// TwinCAT 3 PLC project SPS_Blinker
// ProgramVersion: 3.1.4026.19
// libraries:
//   Tc2_Standard, * (Beckhoff Automation GmbH)
//   Tc2_System, * (Beckhoff Automation GmbH)
//   Tc2_Utilities, * (Beckhoff Automation GmbH)
// project tree:
//   DUTs/ st_Data.TcDUT, ST_MyData.TcDUT, U_Convert.TcDUT, U_Convert_REAL.TcDUT
//   GVLs/ GVL.TcGVL, GVL_Blinker.TcGVL
//   GVLs/Temperaturfuehler/ GVL_Temperatur.TcGVL
//   / PlcTask.TcTTO
//   POUs/ alle_5sekunden.TcPOU, Blinker.TcPOU, LineChart.TcPOU, Line_Chart_array.TcPOU, MAIN.TcPOU, Modbus_Register_lesen.TcPOU, Modbus_Register_schreiben.TcPOU, Systemzeit.TcPOU, TOF_Beispiel.TcPOU
//   POUs/Funktionen_u_Bausteine/ FB_Blinker.TcPOU, FB_RWA_Trend_array.TcPOU
// real-time tasks:
//   TASK PlcTask: cycle T#10ms, priority 20, ADS port 350

CONFIGURATION SPS_Blinker
    RESOURCE PLC ON TwinCAT3
        TASK PlcTask(INTERVAL := T#10ms, PRIORITY := 20);
        PROGRAM MAIN WITH PlcTask : MAIN;
    END_RESOURCE
END_CONFIGURATION

// ---- DUTs/st_Data.TcDUT
TYPE st_Data :
STRUCT
	x	: INT;
	y	: INT;
END_STRUCT
END_TYPE

// ---- DUTs/ST_MyData.TcDUT
TYPE ST_MyData :
STRUCT
	Nr		: DINT;
	Zeit 	: DT;
	Wert 	: INT;
END_STRUCT
END_TYPE

// ---- DUTs/U_Convert.TcDUT
TYPE U_Convert :
UNION
	AsWord: ARRAY[0..1] OF WORD;
	AsReal: REAL;
END_UNION
END_TYPE

// ---- DUTs/U_Convert_REAL.TcDUT
TYPE U_Convert_REAL :
UNION
	AsReal: ARRAY[0..1] OF REAL;
	AsWord: WORD;
END_UNION
END_TYPE

// ---- GVLs/GVL.TcGVL
VAR_GLOBAL
	//Systemzeit
	bValid     			: BOOL := FALSE;
	
	dtsystemTime		: DATE_AND_TIME;
	
	todsystemTime		: TIME_OF_DAY;
	
	sAktuelle_Stunde	: STRING(255);	//Aktuelle Stunde als String
	
	iAktuelle_Stunde	: INT;			//Aktuelle Stunde als INT
	
	sAktuelle_Minute	: STRING(255);	//Aktuelle Minute als String
	
	iAktuelle_Minute	: INT;			//Aktuelle Minute als INT
	
	sAktuelle_Sekunde	: STRING(255);	//Aktuelle Sekunde als String
	
	iAktuelle_Sekunde	: INT;			//Aktuelle Sekunde als INT
	
	//Main
	bStartUpFinish		: BOOL;
END_VAR

// ---- GVLs/GVL_Blinker.TcGVL
VAR_GLOBAL
	rStatus		: REAL;
	bBlink		: BOOL;
END_VAR

// ---- GVLs/Temperaturfuehler/GVL_Temperatur.TcGVL
VAR_GLOBAL
//	rH0_Aussentemp_old	: REAL;	//Aussenfühler H0 Überdachung
	rH0_Aussentemp		: REAL;	//Aussenfühler H0 Überdachung
END_VAR

// ---- POUs/MAIN.TcPOU
PROGRAM MAIN
VAR

END_VAR

Systemzeit();
Blinker();
//Line_Chart_array();

//LineChart();
//TOF_Beispiel();

alle_5sekunden();

END_PROGRAM

// ---- POUs/Systemzeit.TcPOU
PROGRAM Systemzeit
VAR
	fbFB_LocalSystemTime: FB_LocalSystemTime;
	fbGETSYSTEMTIME		: GETSYSTEMTIME;
    sNetID     			: T_AmsNetID := '';
    bEnable    			: BOOL := 1;
    dwCycle    			: DWORD(1..86400) := 5;
    dwOpt      			: DWORD := 1;
    tTimeout   			: TIME := DEFAULT_ADS_TIMEOUT;
	//bValid     		: BOOL := FALSE; GVL
	//dtsystemTime		: DATE_AND_TIME; GVL
	tzID       			: E_TimeZoneID := eTimeZoneID_Invalid;
END_VAR
VAR_INPUT
    systemTime 			: TIMESTRUCT;
END_VAR
VAR_OUTPUT
	
END_VAR

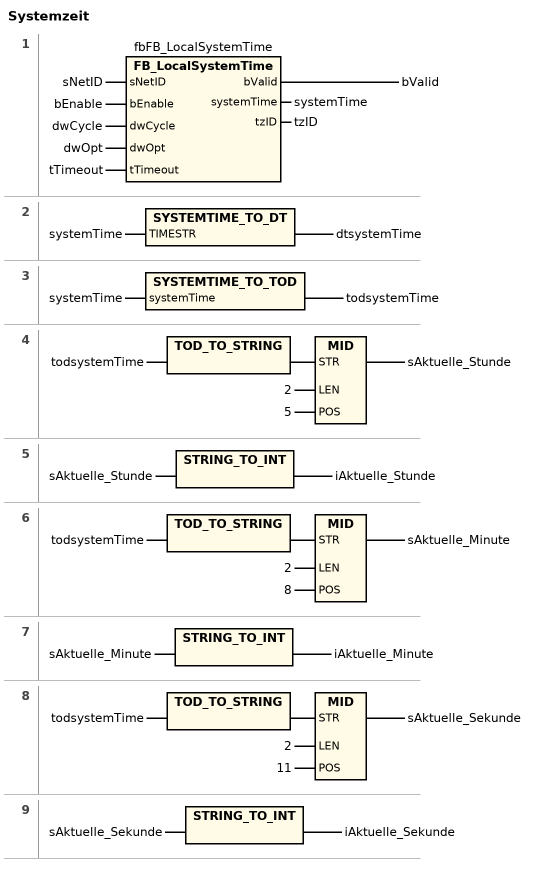
// NETWORK 1
fbFB_LocalSystemTime(
    sNetID := sNetID,
    bEnable := bEnable,
    dwCycle := dwCycle,
    dwOpt := dwOpt,
    tTimeout := tTimeout,
    systemTime => systemTime,
    tzID => tzID); // FB_LocalSystemTime
bValid := fbFB_LocalSystemTime.bValid;

// NETWORK 2
dtsystemTime := SYSTEMTIME_TO_DT(TIMESTR := systemTime);

// NETWORK 3
todsystemTime := SYSTEMTIME_TO_TOD(systemTime := systemTime);

// NETWORK 4
sAktuelle_Stunde := MID(STR := TOD_TO_STRING(todsystemTime), LEN := 2, POS := 5);

// NETWORK 5
iAktuelle_Stunde := STRING_TO_INT(sAktuelle_Stunde);

// NETWORK 6
sAktuelle_Minute := MID(STR := TOD_TO_STRING(todsystemTime), LEN := 2, POS := 8);

// NETWORK 7
iAktuelle_Minute := STRING_TO_INT(sAktuelle_Minute);

// NETWORK 8
sAktuelle_Sekunde := MID(STR := TOD_TO_STRING(todsystemTime), LEN := 2, POS := 11);

// NETWORK 9
iAktuelle_Sekunde := STRING_TO_INT(sAktuelle_Sekunde);

END_PROGRAM

// ---- POUs/Blinker.TcPOU
PROGRAM Blinker
VAR
	fbMyBlinker	: FB_Blinker;
//	bBlink		: BOOL;
END_VAR


fbMyBlinker(tBlinkOn:= T#500MS, tBlinkOff:=T#3S);
bBlink	:= fbMyBlinker.Q;

IF bBlink = TRUE THEN
	rStatus	:= 1;
ELSE	
	rStatus	:= 0;
END_IF

END_PROGRAM

// ---- POUs/Funktionen_u_Bausteine/FB_Blinker.TcPOU
FUNCTION_BLOCK FB_Blinker
VAR_INPUT
	tBlinkOn, tBlinkOff	: TIME;
END_VAR
VAR_OUTPUT
	Q	: BOOL;
END_VAR
VAR
	timerOn, timerOff	: TON;
	nState	: INT;
END_VAR

CASE nState OF
	0:		//Blinker on
		timerOn(IN:= TRUE,	PT:=tBlinkOn);
		Q	:= TRUE;
		IF timerOn.Q THEN
			timerOn(IN:=FALSE);
			nState := 1;
		END_IF
	1:		//Blinker off
		timerOff(IN:=TRUE, PT:=tBlinkOff);
		Q	:= FALSE;
		IF timerOff.Q THEN
			timerOff(IN:=FALSE);
			nState := 0;
		END_IF
END_CASE

END_FUNCTION_BLOCK

// ---- POUs/alle_5sekunden.TcPOU
PROGRAM alle_5sekunden
VAR
    arrData : ARRAY[1..10] OF REAL; // Beispiel-Array
    iSum : REAL;
    iAverage : REAL;
    i : INT;
	
END_VAR

// Summe der Elemente berechnen
iSum := 0;
FOR i := 1 TO 10 DO
    iSum := iSum + arrData[i];
END_FOR

// Durchschnitt berechnen (Division durch die Anzahl der Elemente)
//IF 10 > 0 THEN // Prüfen, ob die Anzahl der Elemente größer als 0 ist
    iAverage := iSum / 10; 
//END_IF

END_PROGRAM

// ---- POUs/Funktionen_u_Bausteine/FB_RWA_Trend_array.TcPOU
FUNCTION_BLOCK FB_RWA_Trend_array
VAR_IN_OUT
	aArray	: ARRAY[0..2,1..1000] OF ST_H2_4_trend_array;	
END_VAR
VAR_INPUT
	bFreigabe			: BOOL;
	rTrueWert			: REAL;
	rFalseWert			: REAL;	
	iArray_i			: DINT := 1;
	bFreigabe_save		: BOOL;	
END_VAR
VAR_OUTPUT
	iArray_i_out		: DINT;
	bFreigabe_save_out	: BOOL;	
END_VAR
VAR
	bEinmallauf			: BOOL;
END_VAR

IF bEinmallauf = FALSE THEN
		IF bFreigabe = TRUE THEN
				aArray[0,iArray_i].Nr	:= iArray_i;	//Laufende Nr
				aArray[0,iArray_i].Zeit	:= dtsystemTime;//Zeit
				aArray[0,iArray_i].Wert	:= rTrueWert;	//Wert Chart
			ELSE
				aArray[0,iArray_i].Nr	:= iArray_i;	//Laufende Nr
				aArray[0,iArray_i].Zeit	:= dtsystemTime;//Zeit
				aArray[0,iArray_i].Wert	:= rFalseWert;	//Wert Chart
		END_IF	
	iArray_i := (iArray_i+1);
	bEinmallauf := TRUE;
END_IF

IF (bFreigabe <> bFreigabe_save) THEN 
		IF bFreigabe = TRUE THEN
				//Zuerst den alten Wert schreiben damit der Chart waagrecht bleibt
				aArray[0,iArray_i].Nr	:= iArray_i;
				aArray[0,iArray_i].Zeit	:= dtsystemTime;
				aArray[0,iArray_i].Wert	:= rFalseWert;
				iArray_i := (iArray_i+1);				
				//Angezeigte Werte
				aArray[0,iArray_i].Nr	:= iArray_i;	//Laufende Nr
				aArray[0,iArray_i].Zeit	:= dtsystemTime;//Zeit
				aArray[0,iArray_i].Wert	:= rTrueWert;	//Wert Chart
			ELSE
				//Zuerst den alten Wert schreiben damit der Chart waagrecht bleibt			
				aArray[0,iArray_i].Nr	:= iArray_i;
				aArray[0,iArray_i].Zeit	:= dtsystemTime;
				aArray[0,iArray_i].Wert	:= rTrueWert;
				iArray_i := (iArray_i+1);				
				//Angezeigte Werte
				aArray[0,iArray_i].Nr	:= iArray_i;	//Laufende Nr
				aArray[0,iArray_i].Zeit	:= dtsystemTime;//Zeit
				aArray[0,iArray_i].Wert	:= rFalseWert;	//Wert Chart
		END_IF
	iArray_i := (iArray_i+1);	
	
	//Zeit wie lannge das array aufgezeichnet werden soll
	IF (dtsystemTime > ((aArray[0,1].Zeit) + T#600M)) THEN
	iArray_i := 1;
	END_IF
	
	bFreigabe_save := bFreigabe;
END_IF

	IF (iAktuelle_Sekunde = 0) OR (iAktuelle_Sekunde = 10) OR (iAktuelle_Sekunde = 20) OR (iAktuelle_Sekunde = 30) OR (iAktuelle_Sekunde = 40) OR (iAktuelle_Sekunde = 50) THEN
		IF (bFreigabe = bFreigabe_save) THEN 
			IF bFreigabe = TRUE THEN				
					//Angezeigte Werte
					aArray[0,iArray_i].Nr	:= iArray_i;	//Laufende Nr
					aArray[0,iArray_i].Zeit	:= dtsystemTime;//Zeit
					aArray[0,iArray_i].Wert	:= rTrueWert;	//Wert Chart
				ELSE				
					//Angezeigte Werte
					aArray[0,iArray_i].Nr	:= iArray_i;	//Laufende Nr
					aArray[0,iArray_i].Zeit	:= dtsystemTime;//Zeit
					aArray[0,iArray_i].Wert	:= rFalseWert;	//Wert Chart
			END_IF
		END_IF
	END_IF
	
	iArray_i_out		:= iArray_i;
	bFreigabe_save_out	:= bFreigabe_save;

END_FUNCTION_BLOCK

// ---- POUs/LineChart.TcPOU
PROGRAM LineChart
VAR
	TestData	: ARRAY[0..1,1..10000] OF st_Data;
	i : INT;
	Test : BOOL;
END_VAR

FOR i := 1 TO 10000 DO
	IF Test THEN
		TestData[0,i].x := i;
		TestData[0,i].y := i;
	ELSE
		TestData[0,i].x := i;
		TestData[0,i].y := 4;			
	END_IF
END_FOR

END_PROGRAM

// ---- POUs/Line_Chart_array.TcPOU
PROGRAM Line_Chart_array
VAR
	TestData						: ARRAY[0..2,1..1000] OF ST_MyData;
	i								: DINT := 1;
	bStatus_array_save				: BOOL;
END_VAR


IF bBlink <> bStatus_array_save THEN 
		IF bBlink = TRUE THEN
				//Zuerst den alten Wert schreiben damit der Chart waagrecht bleibt
				TestData[0,i].Nr	:= i;
				TestData[0,i].Zeit	:= dtsystemTime;
				TestData[0,i].Wert	:= 0;
				i := (i+1);				

				TestData[0,i].Nr	:= i;			//Laufende Nr
				TestData[0,i].Zeit	:= dtsystemTime;//Zeit
				TestData[0,i].Wert	:= 1;			//Wert Chart
			ELSE
				//Zuerst den alten Wert schreiben damit der Chart waagrecht bleibt			
				TestData[0,i].Nr	:= i;
				TestData[0,i].Zeit	:= dtsystemTime;
				TestData[0,i].Wert	:= 1;
				i := (i+1);				

				TestData[0,i].Nr	:= i;			//Laufende Nr
				TestData[0,i].Zeit	:= dtsystemTime;//Zeit
				TestData[0,i].Wert	:= 0;			//Wert Chart
		END_IF
	i := (i+1);
	
	//Zeit wie lannge das array aufgezeichnet werden soll
	IF (dtsystemTime > ((TestData[0,1].Zeit) + T#90M) OR (i > 995)) THEN
	i := 1;
	END_IF
	
	bStatus_array_save := bBlink;
END_IF

END_PROGRAM

// ---- POUs/Modbus_Register_lesen.TcPOU
PROGRAM Modbus_Register_lesen
VAR
	uModbusConvert: U_Convert;	//Union zur Konvertierung
	nWord: ARRAY[0..1] OF WORD;	//Wert, der konvertiert wird
	nDWORD: DWORD;	//Wert, der per Modbus empfangen wird
END_VAR

uModbusConvert.AsWord[0] := GVL_Modbus.mb_Output_Registers[0];	//Zuweisung LowWORD evtl. tauschen
uModbusConvert.AsWord[1] := GVL_Modbus.mb_Output_Registers[0];	//Zuweisung HighWORD
rTemp_RT_H1_O_Robat := uModbusConvert.AsReal;

uModbusConvert.AsWord[0] := GVL_Modbus.mb_Output_Registers[0];	//Zuweisung LowWORD evtl. tauschen
uModbusConvert.AsWord[1] := GVL_Modbus.mb_Output_Registers[1];	//Zuweisung HighWORD
rTemp_RT_H2_Robat := uModbusConvert.AsReal;

uModbusConvert.AsWord[0] := GVL_Modbus.mb_Output_Registers[0];	//Zuweisung LowWORD evtl. tauschen
uModbusConvert.AsWord[1] := GVL_Modbus.mb_Output_Registers[2];	//Zuweisung HighWORD
rTemp_RT_H3_Robat := uModbusConvert.AsReal;

uModbusConvert.AsWord[0] := GVL_Modbus.mb_Output_Registers[0];	//Zuweisung LowWORD evtl. tauschen
uModbusConvert.AsWord[1] := GVL_Modbus.mb_Output_Registers[3];	//Zuweisung HighWORD
rTemp_RT_H4_S_Robat := uModbusConvert.AsReal;

uModbusConvert.AsWord[0] := GVL_Modbus.mb_Output_Registers[0];	//Zuweisung LowWORD evtl. tauschen
uModbusConvert.AsWord[1] := GVL_Modbus.mb_Output_Registers[4];	//Zuweisung HighWORD
rTemp_RT_H4_N_Robat := uModbusConvert.AsReal;

uModbusConvert.AsWord[0] := GVL_Modbus.mb_Output_Registers[0];	//Zuweisung LowWORD evtl. tauschen
uModbusConvert.AsWord[1] := GVL_Modbus.mb_Output_Registers[5];	//Zuweisung HighWORD
rTemp_RT_H8_1_Robat := uModbusConvert.AsReal;

uModbusConvert.AsWord[0] := GVL_Modbus.mb_Output_Registers[0];	//Zuweisung LowWORD evtl. tauschen
uModbusConvert.AsWord[1] := GVL_Modbus.mb_Output_Registers[6];	//Zuweisung HighWORD
rTemp_RT_H8_2_Robat := uModbusConvert.AsReal;

uModbusConvert.AsWord[0] := GVL_Modbus.mb_Output_Registers[0];	//Zuweisung LowWORD evtl. tauschen
uModbusConvert.AsWord[1] := GVL_Modbus.mb_Output_Registers[8];	//Zuweisung HighWORD
rTemp_RT_H8_mittel_Robat := uModbusConvert.AsReal;

uModbusConvert.AsWord[0] := GVL_Modbus.mb_Output_Registers[0];	//Zuweisung LowWORD evtl. tauschen
uModbusConvert.AsWord[1] := GVL_Modbus.mb_Output_Registers[9];	//Zuweisung HighWORD
rH2_3_AK_n_AT_Aus_Anzeige := uModbusConvert.AsReal;

uModbusConvert.AsWord[0] := GVL_Modbus.mb_Output_Registers[0];	//Zuweisung LowWORD evtl. tauschen
uModbusConvert.AsWord[1] := GVL_Modbus.mb_Output_Registers[10];	//Zuweisung HighWORD
rH4_AK_n_AT_Aus_Anzeige := uModbusConvert.AsReal;

END_PROGRAM

// ---- POUs/Modbus_Register_schreiben.TcPOU
PROGRAM Modbus_Register_schreiben
VAR

	uModbusConvert: U_Convert_REAL;	//Union zur Konvertierung
	nReal: ARRAY[0..1] OF REAL;	//Wert, der konvertiert wird
	//nDWORD: DWORD;	//Wert, der per Modbus empfangen wird

	rH0_Aussentemp_Word: DWORD;
END_VAR

(*
uModbusConvert.AsWord[0] := GVL_Modbus.mb_Output_Registers[0];	//Zuweisung LowWORD evtl. tauschen
uModbusConvert.AsWord[1] := GVL_Modbus.mb_Output_Registers[0];	//Zuweisung HighWORD
rTemp_RT_H1_O_Robat := uModbusConvert.AsReal;

16791	=	18.9
16788	=	18.5
16784	=	18
16834	=	24.3

*)

uModbusConvert.AsReal[0] := rH0_Aussentemp;
//uModbusConvert.AsReal[1] := rH0_Aussentemp;
rH0_Aussentemp_Word := uModbusConvert.AsWord;

END_PROGRAM

// ---- POUs/TOF_Beispiel.TcPOU
PROGRAM TOF_Beispiel
VAR
	
	iTest1	: INT	:= 0;
	iTest2	: INT;


	fbTOF 	: TOF;
	bVar1	: BOOL;
	
	bTOFout	: BOOL;
	
	bWind_mittel_temp	: BOOL;
	bWind_mittel		: BOOL;
	tTOF_abgel			: TIME;
END_VAR




IF iTest1 > iTest2 THEN
	bWind_mittel_temp	:= TRUE;
ELSE
	bWind_mittel_temp	:= FALSE;	
END_IF



fbTOF(IN := bWind_mittel_temp, PT := T#5S);
bWind_mittel := fbTOF.Q;
tTOF_abgel	 := fbTOF.ET;





(*
fbTOF(IN := bVar1, PT := T#5S);
bTOFout := fbTOF.Q;
*)

END_PROGRAM
